Fanuc KAREL source: NC0016.KL

-- PROVISIONAL review KL for V1013-1; original PC SHA256 aeffbab0cf676a69651e640b786924bc9952c797e4ba8a1948b12df66633eaf3
-- Incomplete behavior may be omitted. Consult companion uncertainty JSON. Do not deploy.
PROGRAM NC0016
%NOLOCKGROUP
-- UNRESOLVED_LOCAL_POOL 1 cells at code offset 3; source declarations unknown
-- DIRECT_LOCAL_WORD_ACCESS alone does not prove INTEGER, REAL, or BOOLEAN
BEGIN
  -- UNRESOLVED_PC offsets 0-8; opcodes 2B,2C,7B
  -- UNRESOLVED_PC offsets 13-20; opcodes 9D,23
  -- UNRESOLVED_PC offsets 25-38; opcodes 21,9D,57,79
  -- UNRESOLVED_PC offsets 43-61; opcodes 21,2E,52,23
  -- UNRESOLVED_PC offsets 66-71; opcodes 7A
  -- UNRESOLVED_PC offsets 76-89; opcodes 21,9D,57,79
  -- UNRESOLVED_PC offsets 94-112; opcodes 21,2E,52,23
  -- UNRESOLVED_PC offsets 117-122; opcodes 7A
  -- UNRESOLVED_PC offsets 127-140; opcodes 21,9D,57,79
  -- UNRESOLVED_PC offsets 145-163; opcodes 21,2E,52,23
  -- UNRESOLVED_PC offsets 168-173; opcodes 7A
  -- UNRESOLVED_PC offsets 178-191; opcodes 21,9D,57,79
  -- UNRESOLVED_PC offsets 196-214; opcodes 21,2E,52,23
  -- UNRESOLVED_PC offsets 219-224; opcodes 7A
  -- UNRESOLVED_PC offsets 229-242; opcodes 21,9D,57,79
  -- UNRESOLVED_PC offsets 247-265; opcodes 21,2E,52,23
  -- UNRESOLVED_PC offsets 270-275; opcodes 7A
  -- UNRESOLVED_PC offsets 280-293; opcodes 21,9D,57,79
  -- UNRESOLVED_PC offsets 298-316; opcodes 21,2E,52,23
  -- UNRESOLVED_PC offsets 321-326; opcodes 7A
  -- UNRESOLVED_PC offsets 331-344; opcodes 21,9D,57,79
  -- UNRESOLVED_PC offsets 349-367; opcodes 21,2E,52,23
  -- UNRESOLVED_PC offsets 372-377; opcodes 7A
  -- UNRESOLVED_PC offsets 382-395; opcodes 21,9D,57,79
  -- UNRESOLVED_PC offsets 400-418; opcodes 21,2E,52,23
  -- UNRESOLVED_PC offsets 423-428; opcodes 7A
  -- UNRESOLVED_PC offsets 433-447; opcodes 21,9D,52,23
  -- UNRESOLVED_PC offsets 492-496; opcodes 7F
  -- UNRESOLVED_PC offsets 501-505; opcodes 27,AA
  -- UNRESOLVED_PC offsets 510-514; opcodes 7F
END NC0016
